TYPE DInputs :
STRUCT
	input1 : BOOL;
	input2 : BOOL;
	input3 : BOOL;
	input4 : BOOL;
	controlInput1 : BOOL;
	controlInput2 : BOOL;
	controlInput3 : BOOL;
	controlInput4 : BOOL;
END_STRUCT
END_TYPE

(* stored: Version 1.1.0.1, ProductVersion 3.1.4024.11
   DUT DInputs: Id {8277fb9e-1978-47d6-aaed-4f4f4dc3c2aa} *)
